TYPE ST_MoviCPosition_Config :
STRUCT
	pMovisafeCSSx1a			: POINTER TO FB_MovisafeCSSx1a; //[optional] Pointer to a MovisafeCSSx1a instance
	nSoftwareLimitMin		: DINT := -2147483648;	//Position limit minimum in LU
	nSoftwareLimitMax		: DINT := 2147483647;	//Position limit maximum in LU
	nReferencePos			: DINT := 0;			//Reference position in LU when using mode 300
	fDecCoastStop			: REAL := 1000.0;		//Deceleration for coast/brake stop in LU/s^2
	fDecEstop				: REAL := 100.0;		//Deceleration for emergency stop in LU/s^2
	fDecelerationLimit		: REAL := 100.0;		//Decceleration limit (bus stop) in LU/s^2
	fRatioVelocity			: REAL := 1.0;			//Ratio for setpoint velocity
	fRatioAccDec			: REAL := 1.0;			//Ratio for setpoint acceleration/deceleration
	fRatioPosition			: REAL := 1.0;			//Ratio for position output
	nJerk					: INT  := 0;			//Jerk from 0 to 100%
	fPositionOffset			: REAL := 0;
	fInitPosition			: REAL := 0;
	fResolution				: REAL := 0.1;
	bSwapProcessData		: BOOL; //SWAP Process Data from/to FIELDBUS
END_STRUCT
END_TYPE

(* stored: Version 1.1.0.1, ProductVersion 3.1.4024.12
   DUT ST_MoviCPosition_Config: Id {dce56971-73a4-0dea-1b8a-3cf734f38b2d} *)
